(*
	This function block publishes the testresults into a JUnit compatible XmlFile
*)
{attribute 'hide_all_locals'}
FUNCTION_BLOCK FB_JUnitXmlPublisher IMPLEMENTS I_TestResultLogger
VAR     
    (* Dependancy Injection via FB_Init*)
    TestResults : I_TestResults; 
    
    (* path for storing the output file *)
    szFilename : STRING := 'testresults.xml';
    
    (* file access mode *)
    stFileAccessMode : SysFile.ACCESS_MODE := SysFile.AM_WRITE_PLUS;
        
    File : FB_FileControl;
	Xml : FB_XMLControl;
    BufferInitialised : BOOL := FALSE;
	Buffer : ARRAY [0..(GVL_Param_XmlControl.MaxFileSize-1)] OF BYTE;
    WritingTestSuiteResultNumber : UINT(1..GVL_Param_TcUnit.MaxNumberOfTestSuites);
    PublishTrigger : R_TRIG;
END_VAR

(*
    FB_Init is always available implicitly AND it is used primarily FOR initialization.
    The return value is not evaluated. For a specific influence, you can also declare the
    methods explicitly and provide additional code there with the standard initialization
    code. You can evaluate the return value.
*)
METHOD FB_Init: BOOL
VAR_INPUT
    bInitRetains: BOOL; // TRUE: the retain variables are initialized (reset warm / reset cold)
    bInCopyCode: BOOL;  // TRUE: the instance will be copied to the copy code afterward (online change)
    iTestResults : I_TestResults; (* dependency injection *)   
END_VAR
// Set Filepath
szFilename := GVL_Param_XmlControl.FilePath;
// Set buffer and flag
Xml.SetBuffer(pString := ADR(Buffer), iSizeOf := SIZEOF(Buffer));
BufferInitialised := TRUE;

TestResults := iTestResults;
END_METHOD

METHOD PRIVATE Initialised : BOOL
VAR_INPUT
END_VAR
Initialised := THIS^.BufferInitialised;
END_METHOD

(*
    This method is responsible for the entire generation of the testresults.xml output. 
    The output of the xml writer is NOT beautified.
    
    When new data is available, feel free to add it to the report
*)
METHOD PUBLIC LogTestSuiteResults
VAR
    CfUnitTestResults : REFERENCE TO ST_TestSuiteResults;
    CurSuiteNr: UINT;
    CurTestCnt : UINT;
END_VAR
VAR CONSTANT
    TEST_STATUS_SKIP : STRING := 'SKIP';
    TEST_STATUS_PASS : STRING := 'PASS';
    TEST_STATUS_FAIL : STRING := 'FAIL';
END_VAR
CfUnitTestResults REF=TestResults.GetTestSuiteResults();

// Only publish once if "EnablePublish" is enabled and all test results are stored.
PublishTrigger(CLK := (TestResults.GetAreTestResultsAvailable() AND GVL_Param_XmlControl.EnablePublish) );
IF PublishTrigger.Q THEN
          
    (* <?xml version="1.0" encoding="UTF-8"?> *)
    Xml.writeDocumentHeader(Header := '<?xml version="1.0" encoding="UTF-8"?>');
    
    (* <testsuites> *)
    xml.NewTag('testsuites');
    Xml.NewParameter('disabled', '');
    Xml.NewParameter('failures', UINT_TO_STRING(CfUnitTestResults.NumberOfFailedTestCases));
    Xml.NewParameter('tests', UINT_TO_STRING(CfUnitTestResults.NumberOfSuccessfulTestCases));

    FOR CurSuiteNr := 1 TO CfUnitTestResults.NumberOfTestSuites BY 1 DO 
        (* <testsuite> *)
        xml.NewTag('testsuite');
        Xml.NewParameter('id', UINT_TO_STRING(CfUnitTestResults.TestSuiteResults[CurSuiteNr].Identity));
        Xml.NewParameter('name', CfUnitTestResults.TestSuiteResults[CurSuiteNr].name);
        Xml.NewParameter('tests', UINT_TO_STRING(CfUnitTestResults.TestSuiteResults[CurSuiteNr].NumberOfTests));        
        Xml.NewParameter('failures', UINT_TO_STRING(CfUnitTestResults.TestSuiteResults[CurSuiteNr].NumberOfFailedTests));
           
        FOR CurTestCnt := 1 TO CfUnitTestResults.TestSuiteResults[CurSuiteNr].NumberOfTests BY 1 DO
            (* <testcase> *)
            Xml.NewTag('testcase');
            Xml.NewParameter('name', CfUnitTestResults.TestSuiteResults[CurSuiteNr].TestCaseResults[CurTestCnt].TestName);
            Xml.NewParameter('classname', CfUnitTestResults.TestSuiteResults[CurSuiteNr].TestCaseResults[CurTestCnt].TestClassName);
            
            IF CfUnitTestResults.TestSuiteResults[CurSuiteNr].TestCaseResults[CurTestCnt].TestIsFailed THEN
                Xml.NewParameter('status', TEST_STATUS_FAIL);
            ELSIF CfUnitTestResults.TestSuiteResults[CurSuiteNr].TestCaseResults[CurTestCnt].TestIsSkipped THEN   
                Xml.NewParameter('status', TEST_STATUS_SKIP);
            ELSE
                Xml.NewParameter('status', TEST_STATUS_PASS);
			END_IF

            (* determine testcase fail or succes *)
            IF CfUnitTestResults.TestSuiteResults[CurSuiteNr].TestCaseResults[CurTestCnt].FailureType <> E_AssertionType.Type_UNDEFINED THEN 
                (* in case of fail 
                    <failure message="Values differ" type="BYTE" />
                *)
                Xml.NewTag('failure');
                Xml.NewParameter('message', CfUnitTestResults.TestSuiteResults[CurSuiteNr].TestCaseResults[CurTestCnt].FailureMessage );
                Xml.NewParameter('type', F_AssertionTypeToString(CfUnitTestResults.TestSuiteResults[CurSuiteNr].TestCaseResults[CurTestCnt].FailureType) );       
                (* close failure tag*)
                Xml.CloseTag();
                
            ELSE
            (* In case of succes *)
            Xml.NewTagData('');
            
            END_IF
            (* close testcase tag*)         
            Xml.CloseTag();
            
        END_FOR
        (* close testsuite tag *)
        Xml.CloseTag();
        
    END_FOR    
    (* Close testsuites *)
    Xml.CloseTag();

    (* Open, save and close the file *)
    OpenWriteClose();
    
    (* clear the internal buffer *)
    Xml.ClearBuffer();
    
    (* inform user *)
    GVL_TcUnit.AdsMessageQueue.WriteLog(MsgCtrlMask := Tc2_System.ADSLOG_MSGTYPE_HINT,
                                        msgFmtStr := '%s',
                                        strArg := '| ==========EXPORTING XML RESULTS==========='); 
    
    GVL_TcUnit.AdsMessageQueue.WriteLog(MsgCtrlMask := Tc2_System.ADSLOG_MSGTYPE_HINT,
                                        msgFmtStr :=  '| Location: %s ',
                                        strArg := GVL_Param_XmlControl.FilePath);

    GVL_TcUnit.AdsMessageQueue.WriteLog(MsgCtrlMask := Tc2_System.ADSLOG_MSGTYPE_HINT,
                                        MsgFmtStr := '%s',
                                        StrArg := '| ===================================='); 
END_IF
END_METHOD

METHOD PRIVATE OpenWriteClose : SysFile.SysTypes.RTS_IEC_RESULT;
VAR
END_VAR
// Open the file, write buffer and close it
OpenWriteClose := SysDir.CmpErrors.Errors.ERR_OK;
IF Initialised() THEN
    OpenWriteClose := MAX(OpenWriteClose, File.Open(Filename := szFilename, FileAccessMode := stFileAccessMode));
    OpenWriteClose := MAX(OpenWriteClose, File.Write(pString := ADR(Buffer), xml.Length)); 
    OpenWriteClose := MAX(OpenWriteClose, File.Close());
ELSE
    OpenWriteClose := SysDir.CmpErrors.Errors.ERR_NOBUFFER;
END_IF;
END_METHOD

END_FUNCTION_BLOCK

(* stored: Version 1.1.0.1, ProductVersion 3.1.4022.18
   POU FB_JUnitXmlPublisher: Id {6597c0b3-0890-4d5d-8d3a-2d0d0b2355db}, SpecialFunc None
   Method FB_Init: Id {0f23c47b-7245-415e-b489-0ae429217263}
   Method Initialised: Id {dac11801-83e2-4726-b3a7-dcd7f73621e3}
   Method LogTestSuiteResults: Id {32c3ccd7-3470-4554-b54c-b3a0a6491553}
   Method OpenWriteClose: Id {84256533-6eb5-465b-b1e5-db6f61e2e6c3} *)
